FUNCTION_BLOCK Conveyor2Check (* Template for a Basic Function Block Type *)
  (* Standard: 61499-2 *)
  (* Version 1.0, 2021-07-28, Tuojian Lyu *)
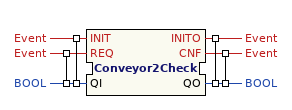
  EVENT_INPUT
    INIT WITH QI; (* Initialization Request *)
    REQ WITH QI; (* Normal Execution Request *)
  END_EVENT
  EVENT_OUTPUT
    INITO WITH QO; (* Initialization Confirm *)
    CNF WITH QO; (* Execution Confirmation *)
  END_EVENT
  VAR_INPUT
    QI : BOOL; (* Input event qualifier *)
  END_VAR
  VAR_OUTPUT
    QO : BOOL; (* Output event qualifier *)
  END_VAR
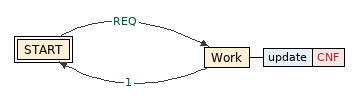
  EC_STATES
    START; (* Initial State *)
    Work : update -> CNF;
  END_STATES
  EC_TRANSITIONS
    START TO Work := REQ;
    Work TO START := 1;
  END_TRANSITIONS
  ALGORITHM update IN ST:
IF TRUE = QI THEN
QO := FALSE;
ELSE
QO := TRUE;
END_IF;
  END_ALGORITHM
END_FUNCTION_BLOCK
